FUNCTION_BLOCK PAEScrew EXTENDS PAETransport
VAR_INPUT
END_VAR
VAR_OUTPUT
END_VAR
VAR
END_VAR

END_FUNCTION_BLOCK

(* stored: Version 1.1.0.1, ProductVersion 3.1.4020.12
   POU PAEScrew: Id {9472cbb9-9085-4b47-8d27-6812fb4a4a62}, SpecialFunc None *)
